INTERFACE Temp_ITFLoopband

METHOD Beweeg
VAR_INPUT
END_VAR
END_METHOD

METHOD BeweegInLift
VAR_INPUT
END_VAR
END_METHOD

METHOD Stop
VAR_INPUT
END_VAR
END_METHOD

END_INTERFACE

(* stored: Version 1.1.0.1
   Itf Temp_ITFLoopband: Id {76e35b7f-ed7b-4848-936f-3291c0e677ac}
   Method Beweeg: Id {ab9487de-8c7f-4ff0-bb0c-695973b98961}
   Method BeweegInLift: Id {61375354-0863-4f64-a6ca-a9d5949a13c3}
   Method Stop: Id {73cfbbd7-6a2b-4600-b4f3-94fca7ba01b8} *)
